TYPE UDT_Scara :
STRUCT
	i: UDT_Scara_DI;
	o: UDT_Scara_DO;
	Busy: BOOL;
	DI_: ARRAY[1..8] OF ARRAY[1..8] OF BOOL;
	DO_: ARRAY[1..8] OF ARRAY[1..8] OF BOOL;
END_STRUCT
END_TYPE

(* stored: Version 1.1.0.1, ProductVersion 3.1.4022.16
   DUT UDT_Scara: Id {e48fa406-374b-43b1-886b-4341820061a7} *)
